// TIA Portal V19 export
TYPE "LEXCHANGETRAY_typeSR1000ProcessValues"
// simulated: Bool
// busyStatusBits: LEXCHANGETRAY_typeSr1000ProfinetTelegram_busyStatusBits
// completionStatusBits: LEXCHANGETRAY_typeSr1000ProfinetTelegram_completionStatusBits
// errorStatusBits: LEXCHANGETRAY_typeSr1000ProfinetTelegram_errorStatusBits
// handshakAndGeneralErrorStatusBits: LEXCHANGETRAY_typeSr1000ProfinetTelegram_handshakAndGeneralErrorStatusBits
// matchingLevelandTotalEvaluationGradeStatus: LEXCHANGETRAY_typeSr1000ProfinetTelegram_matchingLevelandTotalEvaluationGradeStatus
// operationResultStatus: LEXCHANGETRAY_typeSr1000ProfinetTelegram_operationResultStatus
// terminalStatusBits: LEXCHANGETRAY_typeSr1000ProfinetTelegram_terminalStatusBits
// unstableReadStatusBits: LEXCHANGETRAY_typeSr1000ProfinetTelegram_unstableReadStatusBits
// readData128Byte: LEXCHANGETRAY_typeSr1000ProfinetTelegram_readData128Byte
// code: String
// error: Bool
// complete: Bool
// stored: Access Published
   STRUCT
      simulated : Bool;
      busyStatusBits : "LEXCHANGETRAY_typeSr1000ProfinetTelegram_busyStatusBits";
      completionStatusBits { S7_SetPoint := 'True'} : "LEXCHANGETRAY_typeSr1000ProfinetTelegram_completionStatusBits";
      errorStatusBits { S7_SetPoint := 'True'} : "LEXCHANGETRAY_typeSr1000ProfinetTelegram_errorStatusBits";
      handshakAndGeneralErrorStatusBits { S7_SetPoint := 'True'} : "LEXCHANGETRAY_typeSr1000ProfinetTelegram_handshakAndGeneralErrorStatusBits";
      matchingLevelandTotalEvaluationGradeStatus { S7_SetPoint := 'True'} : "LEXCHANGETRAY_typeSr1000ProfinetTelegram_matchingLevelandTotalEvaluationGradeStatus";
      operationResultStatus { S7_SetPoint := 'True'} : "LEXCHANGETRAY_typeSr1000ProfinetTelegram_operationResultStatus";
      terminalStatusBits { S7_SetPoint := 'True'} : "LEXCHANGETRAY_typeSr1000ProfinetTelegram_terminalStatusBits";
      unstableReadStatusBits { S7_SetPoint := 'True'} : "LEXCHANGETRAY_typeSr1000ProfinetTelegram_unstableReadStatusBits";
      readData128Byte { S7_SetPoint := 'True'} : "LEXCHANGETRAY_typeSr1000ProfinetTelegram_readData128Byte";
      code { S7_SetPoint := 'True'} : String;
      error { S7_SetPoint := 'True'} : Bool;   // 扫码结果报错
      complete : Bool;   // 扫码完毕包含重试
   END_STRUCT;
END_TYPE
